FUNCTION_BLOCK Measurement IMPLEMENTS IOut
VAR_INPUT
    value : LREAL;
END_VAR
VAR
    _out : LREAL;
END_VAR

_out := value;

METHOD Derivative : REFERENCE TO Measurement
VAR_INPUT
END_VAR
END_METHOD

PROPERTY Out : LREAL
GET
OUT := _out;
END_GET
END_PROPERTY

END_FUNCTION_BLOCK

(* stored: Version 1.1.0.1, ProductVersion 3.1.4024.12
   POU Measurement: Id {d5e65a98-c59a-40a4-8e08-14b2a0104701}, SpecialFunc None
   Method Derivative: Id {3cb626dd-f306-4dd7-8b41-c5d14146e141}
   Property Out: Id {f11c0c9d-cbae-4516-9e11-e42329123126}
   Get Get: Id {42b506ae-6bce-45b3-bdd7-aeb51ebf09f3} *)
